{attribute 'linkalways'} 
{attribute 'no_explicit_call' := 'This FB is a CLASS and must be accessed using methods or properties'}
{attribute 'enable_dynamic_creation'}
FUNCTION_BLOCK EnumDatatypeAddedEvent EXTENDS Disposable IMPLEMENTS I_EnumDatatypeAddedEvent
VAR
	_target : I_EnumDatatype;
END_VAR

METHOD FB_init : BOOL
VAR_INPUT
	bInitRetains : BOOL; // if TRUE, the retain variables are initialized (warm start / cold start)
	bInCopyCode : BOOL;  // if TRUE, the instance afterwards gets moved into the copy code (online change)
	Target : I_EnumDatatype;
END_VAR
This^._target := Target;
END_METHOD

PROPERTY PUBLIC Target : I_EnumDatatype
GET
Target := _target;
END_GET
END_PROPERTY

END_FUNCTION_BLOCK

(* stored: Version 1.1.0.1, ProductVersion 3.1.4024.12
   POU EnumDatatypeAddedEvent: Id {bff7a8fa-a624-0127-38a3-cd4031d2f5d2}, SpecialFunc None
   Folder Constructor: Id {6bad2482-2c6a-0dbc-115a-2a0eeade0273}
   Method FB_init: Id {2e42f182-e43d-0232-22c0-52369e1af156}
   Property Target: Id {b17a6e2e-3337-0fc0-3c1d-8bac96d8f35a}
   Get Get: Id {7ee46344-83f5-089c-074d-5321cdfda7c7} *)
